PROGRAM MAIN
VAR
END_VAR

END_PROGRAM

(* stored: Version 1.1.0.1
   POU MAIN: Id {0eabfe41-4ae4-4ad9-b199-1cf6ff8d2d43} *)
